RoboDK station: STATION.rdk

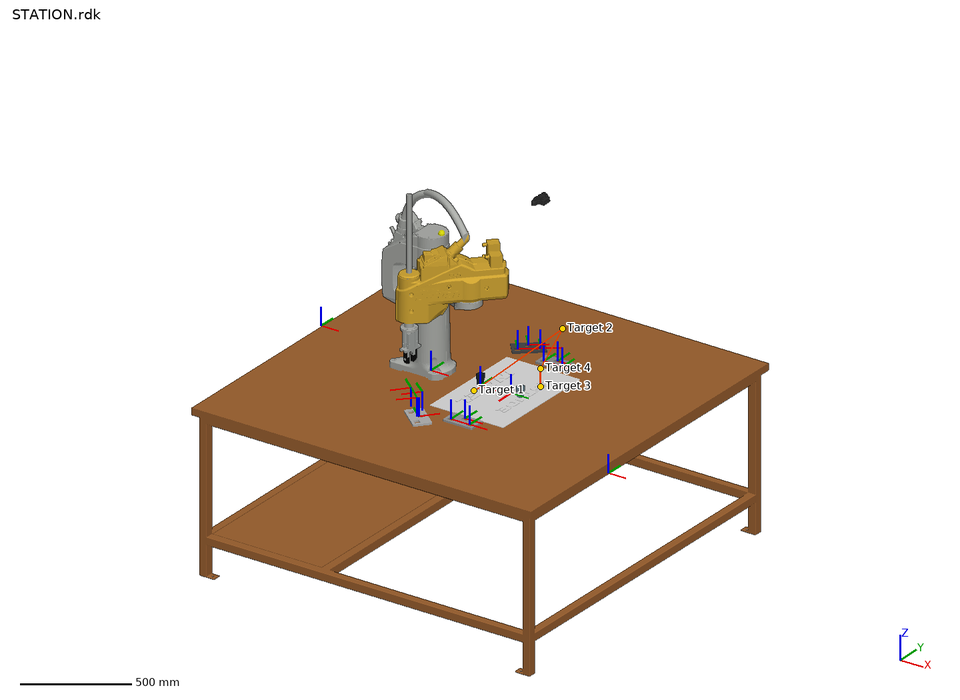
[picture v0: the station drawn from its stored meshes, robots at their saved joint values, targets as dots, program paths as lines]
Station STATION testes Guilherme  (saved by RoboDK 5.7.0). Poses are relative to the parent item; angles as X-Y-Z fixed-axis rotations.
Station parameters (name, value as stored): IO_0, 0
  - object Mesa at (0, 0, 0) mm, size 1850 x 1850 x 835 mm, geometry from Mesa.stl
  - frame Centro Mesa at (0, 0, 835) mm
    - frame Staubli TS60 FL 200 Base at (-267.5, 3, 0) mm
      - robot Staubli TS60 FL 200 (model Staubli TS60 FL 400): 4 axes, payload 2 kg, reach 600 mm, repeatability 0.01 mm, weight 55 kg
          modified DH rows (alpha deg, a mm, theta deg, d mm): 0, 0, 0, 0; 0, 330, 0, 0; 0, 270, 0, 170 linear; 180, 0, 0, 0
          joint limits [-140, -150, 0, -500] to [140, 150, 200, 500]; home [0, 0, 0, 0]; saved at [-24.862, -109.061, 196.998, -174.229]
        - tool GarraCompleta, TCP at (0, 0, 190) mm, size 97 x 40 x 153.1 mm
    - object SWPart at (-65.5, 303, 0) mm, rotated rx 0 ry 0 rz -90 deg, size 600 x 400 x 6 mm, geometry from Mesabranca.sld
    - object Berco 1 at (-124, -416, 0) mm, rotated rx 0 ry 0 rz -40 deg, size 158 x 89.5 x 10 mm, geometry from Gabarito_TicTac.STL
    - object Berco 2 at (72.5, -395, 0) mm, size 158 x 89.5 x 10 mm, geometry from Gabarito_TicTac.STL
    - object Berco 3 at (72.5, 323.99, 0) mm, size 158 x 89.5 x 10 mm, geometry from Gabarito_TicTac.STL
    - object Berco 4 at (-66.99, 344, 0) mm, rotated rx 0 ry 0 rz 40 deg, size 158 x 89.5 x 10 mm, geometry from Gabarito_TicTac.STL
    - frame Frame Camera at (-930, 90, 0) mm
      - object OpenCV OAK-D Camera at (1190, 0, 950) mm, rotated rx -180 ry 0 rz -90 deg, size 110 x 54.5 x 33 mm, geometry from OpenCV-OAK-D-Camera.sld
    - object Cubo Negro at (1.07, 1.24, 60) mm, rotated rx 180 ry 0 rz 0 deg, size 26 x 26 x 55 mm, geometry from Cubo3_TicTac.STL
    - object Cubo Cinza at (220, 0, 60) mm, rotated rx 180 ry 0 rz 0 deg, size 26 x 26 x 55 mm, geometry from Cubo3_TicTac.STL
    - frame Frame_Centro_Mesa at (163.03, 8.96, 3) mm, rotated rx 0 ry 0 rz -90 deg
      - target Target 1 (Cartesian target) at (354.12, 45.98, 167) mm, rotated rx 180 ry 0 rz 53.68 deg; joints [-26.76, -20.9, 190, -11.34] of Staubli TS60 FL 200
      - target Target 2 (Cartesian target) at (-389.51, 7.51, 167) mm, rotated rx 180 ry 0 rz 131.91 deg; joints [51.47, -20.9, 190, -11.34] of Staubli TS60 FL 200
      - target Target 3 (Cartesian target) at (-0.29, 159.59, 78.81) mm, rotated rx 180 ry 0 rz -10.9 deg; joints [10, -20.9, 101.81, 90] of Staubli TS60 FL 200
      - target Target 4 (Cartesian target) at (-0.29, 159.59, 167) mm, rotated rx 180 ry 0 rz -10.9 deg; joints [10, -20.9, 190, 90] of Staubli TS60 FL 200
    - frame Frame 5 at (-30.26, -429.3, 10) mm, rotated rx 0 ry -0.14 rz 51.21 deg
      - frame centro B2 at (13.27, 0, 120) mm, rotated rx 180 ry 0 rz 180 deg
  - camera Camera 1
  - program Prog1 (7 instructions, listed below)
  - program ProgGui (14 instructions, listed below)
  - frame Centro B1_S1 at (-86.48, -414.85, 965) mm, rotated rx -180 ry 0 rz -130 deg
  - frame Centro B1 S3 at (-8.02, -480.03, 965) mm, rotated rx -180 ry 0 rz -130 deg
  - frame Centro B2  S1 at (0, 1000, 0) mm
  - frame Centro B2 S2 at (151.5, -331, 845) mm
  - frame Centro B2 S3 at (203.06, -368.54, 845) mm
  - frame Centro B2 S1 at (100.5, -369.5, 845) mm
  - frame Centro B4 S1  at (-62.49, 381.16, 845) mm, rotated rx 0 ry 0 rz 40 deg
  - frame Centro B4 S3 at (16.02, 448.2, 845) mm, rotated rx 0 ry 0 rz 40 deg
  - frame Centro B3 S1  at (100.5, 349.49, 845) mm
  - frame Centro B3 S2 at (151.5, 387.99, 845) mm
  - frame Centro B3 S3 at (202.5, 349.49, 845) mm
  - frame Centro B4 S2 at (-47.61, 443.81, 845) mm, rotated rx 0 ry 0 rz 40 deg
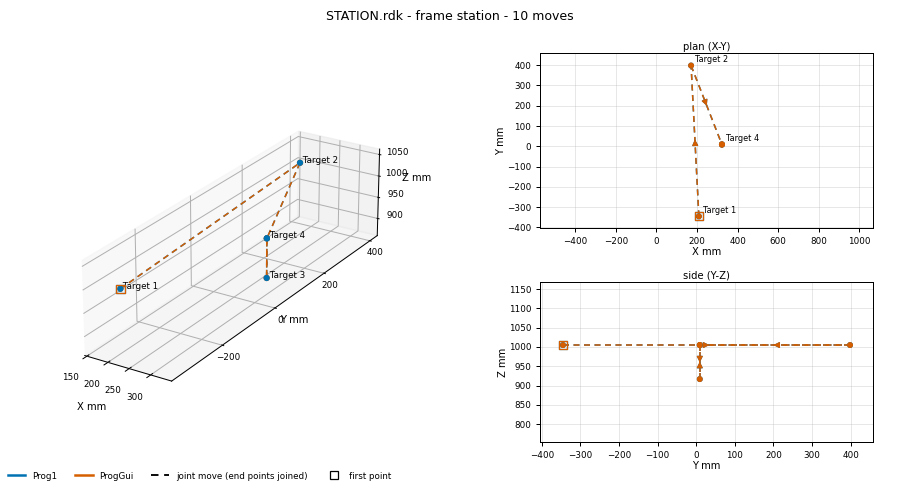
[picture p0: tool path of STATION.rdk in frame station, 10 of 10 moves have a stored position in this frame; points joined in program order, loops and branches not executed]

--- program Prog1 (robot Staubli TS60 FL 200) ---
  Set Ref.: Frame_Centro_Mesa
  Set Tool: GarraCompleta
  MoveJ (Target 1)
  MoveJ (Target 2)
  MoveJ (Target 4)
  MoveJ (Target 3)
  MoveJ (Target 4)

--- program ProgGui (robot Staubli TS60 FL 200) ---
  Set Ref.: Frame_Centro_Mesa
  Set Tool: GarraCompleta
  Set IO_0=0
  Pause 500 ms
  MoveJ (Target 1)
  MoveJ (Target 2)
  MoveJ (Target 4)
  MoveJ (Target 3)
  Set IO_0=1
  Pause 500 ms
  MoveJ (Target 4)
  Set IO_0=0
  Pause 500 ms
  Set speed (45.0 mm/s)
